TYPE ST_MachinePondErrors :
STRUCT
	FeedingPulp							: ST_CilinderErrors;
END_STRUCT
END_TYPE

(* stored: Version 1.1.0.1, ProductVersion 3.1.4020.12
   DUT ST_MachinePondErrors: Id {0454eed2-aea2-4fdb-9c58-1f087006c411} *)
